(* Logix 5000 project; controller SolisPLC_Vlad_CGL1 vendor 1 type 14 code 226 rev 36.11; software revision 36.00 *)

TASK MainTask (continuous, watchdog 500 ms) : MainProgram, DataLink, Palletizer, Tutorials, Communication, SimulatedMachine_v1_0
TASK SafetyTask (periodic, rate 20 ms, priority 10, watchdog 20 ms, safety) : SafetyProgram

MODULES
   Local : vendor 1 type 14 code 226 (5069 0, rev 36.11)
      VFD_07 : PowerFlex 525-EENET (Ethernet 192.168.1.7, rev 1.3, Output RPI 20 ms)
END_MODULES

TYPE Asset_Data_v01_01 :
STRUCT
   machineState : INT;   // The state of the machine - 0 - Unknown State 1 - Running 2 - Stopped 3 - Stopped - Faulted 4 - Running - Starved 5 - Running - Backed-Up
   heartBeat : BOOL;   // A pulse which indicates that the communication with the machine is UP. The pulse is 1 sec ON / 1 sec OFF.
   currentProductionSpeed : INT;   // A count of finished products for the last hour.
END_STRUCT
END_TYPE

TYPE Motor_PF525_Params :
STRUCT
   Param_1_64 : INT[128];
   Param_65_128 : INT[128];
   Param_129_192 : INT[128];
   Param_193_256 : INT[128];
   Param_257_320 : INT[128];
   Param_321_384 : INT[128];
   Param_385_448 : INT[128];
   Param_449_512 : INT[128];
   Param_513_576 : INT[128];
   Param_577_640 : INT[128];
   Param_641_704 : INT[128];
   Param_705_768 : INT[128];
END_STRUCT
END_TYPE

TYPE UDT_MQTT_DINT :
STRUCT
   Message : DINT;
   Delay : DINT;
   Timer : TIMER;
   RawData : DINT;
   Delta : DINT;
   OldRawData : DINT;
END_STRUCT
END_TYPE

TYPE UDT_paramReadReqs :
STRUCT
   Param_1_64 : INT[128];
   Param_65_128 : INT[128];
   Param_129_192 : INT[128];
   Param_193_256 : INT[128];
   Param_257_320 : INT[128];
   Param_321_384 : INT[128];
   Param_385_448 : INT[128];
   Param_449_512 : INT[128];
   Param_513_576 : INT[128];
   Param_577_640 : INT[128];
   Param_641_704 : INT[128];
   Param_705_768 : INT[128];
END_STRUCT
END_TYPE

TYPE udtVariableSpeedMotor :
STRUCT
   Auto : BOOL;   // Auto Mode from RSView
   Interlock : BOOL;   // Pump Run Interlock
   Fault : BOOL;   // Pump Fault
   Start : BOOL;   // Manual Start from RSView
   Stop : BOOL;   // Manual Stop from RSView
   Run : BOOL;   // Drive Run Output Command
   Running : BOOL;   // Running Feedback
   LDS : BOOL;   // Local Disconnect Switch
   FwdCmd : BOOL;   // Run Drive Forward Request
   RevCmd : BOOL;   // Run Drive Reverse Request
   ClearFaults : BOOL;   // Drive Fault Reset Request
   Ready : BOOL;   // Drive Ready Feedback
   FwdAct : BOOL;   // Drive in Run Forward Mode
   RevAct : BOOL;   // Drive in Run Reverse Mode
   Alarm : BOOL;   // Drive Alarm
   DriveFault : BOOL;   // Drive Fault
   AtSpeed : BOOL;   // Drive is At Speed
   APerm : BOOL[32];   // Auto Run Permissive
   FaultTimer : TIMER;   // Start/Stop Timeout
   SpeedSP : REAL;   // Speed Setpoint from RSView
   SpeedSPmin : REAL;   // Speed Setpoint Minimum Limit
   SpeedSPmax : REAL;   // Speed Setpoint Maximum Limit
   SpeedAct : REAL;   // Actual Speed to RSView
   Status : DINT[5];
   Avl : BOOL[32];
   Name : Varchar40;
END_STRUCT
END_TYPE

TYPE Varchar40 :   // String Of 40 Characters
STRUCT
   LEN : DINT;
   DATA : SINT[40];
END_STRUCT
END_TYPE

ADD_ON_INSTRUCTION _AOI_Fah_to_Cel   (* revision 1.0 *)
VAR_INPUT
   Temperature_Fah : REAL; {required}
END_VAR
VAR_OUTPUT
   Temperature_Cel : REAL; {required}
END_VAR
VAR
   Placeholder : REAL; {access None}
   Placeholder1 : REAL; {access None}
END_VAR

ROUTINE Logic   (* ladder *)
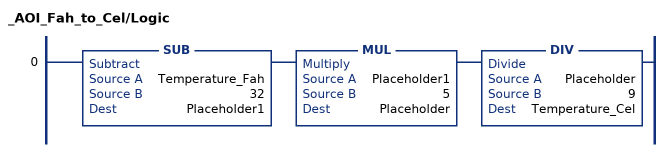
   0: SUB(Temperature_Fah,32,Placeholder1)MUL(Placeholder1,5,Placeholder)DIV(Placeholder,9,Temperature_Cel);
END_ROUTINE
END_ADD_ON_INSTRUCTION

ADD_ON_INSTRUCTION AOI_PF525_GetParam   (* revision 1.0 *)

ROUTINE Logic   (* ladder *)
END_ROUTINE
END_ADD_ON_INSTRUCTION

VAR_GLOBAL   (* controller tags *)
   BOOL_IN_0 : BOOL;
   BOOL_IN_1 : BOOL;   // System Stop PB
   BOOL_OUT_0 : BOOL;   // STATUS - System Running
   BOOL_OUT_1 : BOOL := 1;   // STATUS - System Stopped
   getParam : INT[10];
   M07_Params : Motor_PF525_Params := (Param_1_64[0] := 1, Param_1_64[2] := 2, Param_1_64[4] := 3, Param_1_64[6] := 4, Param_1_64[8] := 5, Param_1_64[9] := 329, Param_1_64[10] := 6, Param_1_64[11] := 2, Param_1_64[12] := 7, Param_1_64[13] := 73, Param_1_64[14] := 8, Param_1_64[15] := 4, Param_1_64[16] := 9, Param_1_64[17] := 73, Param_1_64[18] := 10, Param_1_64[20] := 11, Param_1_64[22] := 12, Param_1_64[23] := 155, Param_1_64[24] := 13, Param_1_64[25] := 1, Param_1_64[26] := 14, Param_1_64[28] := 15, Param_1_64[30] := 16, Param_1_64[32] := 17, Param_1_64[34] := 18, Param_1_64[36] := 19, Param_1_64[38] := 20, Param_1_64[40] := 21, Param_1_64[42] := 22, Param_1_64[44] := 23, Param_1_64[45] := 8, Param_1_64[46] := 24, Param_1_64[48] := 25, Param_1_64[50] := 26, Param_1_64[52] := 27, Param_1_64[53] := 30, Param_1_64[54] := 28, Param_1_64[55] := 53, Param_1_64[56] := 29, Param_1_64[57] := 7001, Param_1_64[58] := 30, Param_1_64[59] := 1, Param_1_64[60] := 31, Param_1_64[61] := 230, Param_1_64[62] := 32, Param_1_64[63] := 60, Param_1_64[64] := 33, Param_1_64[65] := 25, Param_1_64[66] := 34, Param_1_64[67] := 17, Param_1_64[68] := 35, Param_1_64[69] := 4, Param_1_64[70] := 36, Param_1_64[71] := 1750, Param_1_64[72] := 37, Param_1_64[73] := 40, Param_1_64[74] := 38, Param_1_64[76] := 39, Param_1_64[77] := 1, Param_1_64[78] := 40,
        Param_1_64[80] := 41, Param_1_64[81] := 1000, Param_1_64[82] := 42, Param_1_64[83] := 1000, Param_1_64[84] := 43, Param_1_64[86] := 44, Param_1_64[87] := 6000, Param_1_64[88] := 45, Param_1_64[90] := 46, Param_1_64[91] := 5, Param_1_64[92] := 47, Param_1_64[93] := 15, Param_1_64[94] := 48, Param_1_64[95] := 2, Param_1_64[96] := 49, Param_1_64[97] := 5, Param_1_64[98] := 50, Param_1_64[99] := 5, Param_1_64[100] := 51, Param_1_64[101] := 15, Param_1_64[102] := 52, Param_1_64[104] := 53, Param_1_64[106] := 54, Param_1_64[108] := 55, Param_1_64[110] := 56, Param_1_64[112] := 57, Param_1_64[114] := 58, Param_1_64[116] := 59, Param_1_64[118] := 60, Param_1_64[120] := 61, Param_1_64[122] := 62, Param_1_64[123] := 48, Param_1_64[124] := 63, Param_1_64[125] := 50, Param_1_64[126] := 64, Param_65_128[0] := 65, Param_65_128[2] := 66, Param_65_128[3] := 7, Param_65_128[4] := 67, Param_65_128[5] := 5, Param_65_128[6] := 68, Param_65_128[7] := 9, Param_65_128[8] := 69, Param_65_128[9] := 2, Param_65_128[10] := 70, Param_65_128[12] := 71, Param_65_128[14] := 72, Param_65_128[15] := 1, Param_65_128[16] := 73, Param_65_128[18] := 74, Param_65_128[20] := 75, Param_65_128[22] := 76, Param_65_128[24] := 77, Param_65_128[26] := 78, Param_65_128[28] := 79, Param_65_128[30] := 80, Param_65_128[32] := 81, Param_65_128[33] := 13, Param_65_128[34] := 82, Param_65_128[36] := 83,
        Param_65_128[38] := 84, Param_65_128[40] := 85, Param_65_128[42] := 86, Param_65_128[43] := 200, Param_65_128[44] := 87, Param_65_128[45] := 200, Param_65_128[46] := 88, Param_65_128[48] := 89, Param_65_128[49] := 100, Param_65_128[50] := 90, Param_65_128[52] := 91, Param_65_128[54] := 92, Param_65_128[55] := 1000, Param_65_128[56] := 93, Param_65_128[58] := 94, Param_65_128[60] := 95, Param_65_128[62] := 96, Param_65_128[63] := 1000, Param_65_128[64] := 97, Param_65_128[66] := 98, Param_65_128[68] := 99, Param_65_128[70] := 100, Param_65_128[72] := 101, Param_65_128[73] := 100, Param_65_128[74] := 102, Param_65_128[76] := 103, Param_65_128[77] := 150, Param_65_128[78] := 104, Param_65_128[80] := 105, Param_65_128[82] := 106, Param_65_128[84] := 107, Param_65_128[86] := 108, Param_65_128[88] := 109, Param_65_128[90] := 110, Param_65_128[92] := 111, Param_65_128[94] := 112, Param_65_128[96] := 113, Param_65_128[98] := 114, Param_65_128[100] := 115, Param_65_128[102] := 116, Param_65_128[104] := 117, Param_65_128[106] := 118, Param_65_128[108] := 119, Param_65_128[110] := 120, Param_65_128[112] := 121, Param_65_128[114] := 122, Param_65_128[116] := 123, Param_65_128[117] := 3, Param_65_128[118] := 124, Param_65_128[119] := 100, Param_65_128[120] := 125, Param_65_128[122] := 126, Param_65_128[123] := 50, Param_65_128[124] := 127, Param_65_128[126] := 128, Param_65_128[127] := 1, Param_129_192[0] := 129, Param_129_192[1] := 192, Param_129_192[2] := 130, Param_129_192[3] := 168,
        Param_129_192[4] := 131, Param_129_192[5] := 1, Param_129_192[6] := 132, Param_129_192[7] := 7, Param_129_192[8] := 133, Param_129_192[9] := 255, Param_129_192[10] := 134, Param_129_192[11] := 255, Param_129_192[12] := 135, Param_129_192[13] := 255, Param_129_192[14] := 136, Param_129_192[16] := 137, Param_129_192[18] := 138, Param_129_192[20] := 139, Param_129_192[22] := 140, Param_129_192[24] := 141, Param_129_192[26] := 142, Param_129_192[28] := 143, Param_129_192[30] := 144, Param_129_192[32] := 145, Param_129_192[34] := 146, Param_129_192[36] := 147, Param_129_192[38] := 148, Param_129_192[40] := 149, Param_129_192[42] := 150, Param_129_192[44] := 151, Param_129_192[46] := 152, Param_129_192[48] := 153, Param_129_192[49] := 82, Param_129_192[50] := 154, Param_129_192[52] := 155, Param_129_192[54] := 156, Param_129_192[56] := 157, Param_129_192[57] := 14, Param_129_192[58] := 158, Param_129_192[60] := 159, Param_129_192[62] := 160, Param_129_192[64] := 161, Param_129_192[66] := 162, Param_129_192[68] := 163, Param_129_192[70] := 164, Param_129_192[72] := 165, Param_129_192[74] := 166, Param_129_192[76] := 167, Param_129_192[78] := 168, Param_129_192[80] := 169, Param_129_192[82] := 170, Param_129_192[84] := 171, Param_129_192[85] := 2, Param_129_192[86] := 172, Param_129_192[87] := 3, Param_129_192[88] := 173, Param_129_192[89] := 4, Param_129_192[90] := 174, Param_129_192[91] := 5, Param_129_192[92] := 175, Param_129_192[94] := 176, Param_129_192[96] := 177, Param_129_192[98] := 178, Param_129_192[100] := 179,
        Param_129_192[102] := 180, Param_129_192[103] := 241, Param_129_192[104] := 181, Param_129_192[105] := 241, Param_129_192[106] := 182, Param_129_192[107] := 241, Param_129_192[108] := 183, Param_129_192[109] := 241, Param_129_192[110] := 184, Param_129_192[111] := 241, Param_129_192[112] := 185, Param_129_192[113] := 241, Param_129_192[114] := 186, Param_129_192[115] := 241, Param_129_192[116] := 187, Param_129_192[117] := 241, Param_129_192[118] := 188, Param_129_192[120] := 189, Param_129_192[122] := 190, Param_129_192[123] := 300, Param_129_192[124] := 191, Param_129_192[125] := 300, Param_129_192[126] := 192, Param_129_192[127] := 300, Param_193_256[0] := 193, Param_193_256[1] := 300, Param_193_256[2] := 194, Param_193_256[3] := 300, Param_193_256[4] := 195, Param_193_256[5] := 300, Param_193_256[6] := 196, Param_193_256[7] := 300, Param_193_256[8] := 197, Param_193_256[9] := 300, Param_193_256[10] := 198, Param_193_256[12] := 199, Param_193_256[14] := 200, Param_193_256[16] := 201, Param_193_256[18] := 202, Param_193_256[20] := 203, Param_193_256[22] := 204, Param_193_256[24] := 205, Param_193_256[26] := 206, Param_193_256[28] := 207, Param_193_256[30] := 208, Param_193_256[32] := 209, Param_193_256[34] := 210, Param_193_256[36] := 211, Param_193_256[38] := 212, Param_193_256[40] := 213, Param_193_256[42] := 214, Param_193_256[44] := 215, Param_193_256[46] := 216, Param_193_256[48] := 217, Param_193_256[50] := 218, Param_193_256[52] := 219, Param_193_256[54] := 220, Param_193_256[56] := 221, Param_193_256[58] := 222, Param_193_256[60] := 223,
        Param_193_256[62] := 224, Param_193_256[64] := 225, Param_193_256[66] := 226, Param_193_256[68] := 227, Param_193_256[70] := 228, Param_193_256[72] := 229, Param_193_256[74] := 230, Param_193_256[76] := 231, Param_193_256[78] := 232, Param_193_256[80] := 233, Param_193_256[82] := 234, Param_193_256[84] := 235, Param_193_256[86] := 236, Param_193_256[88] := 237, Param_193_256[90] := 238, Param_193_256[92] := 239, Param_193_256[94] := 240, Param_193_256[96] := 241, Param_193_256[98] := 242, Param_193_256[100] := 243, Param_193_256[102] := 244, Param_193_256[104] := 245, Param_193_256[106] := 246, Param_193_256[108] := 247, Param_193_256[110] := 248, Param_193_256[112] := 249, Param_193_256[114] := 250, Param_193_256[116] := 251, Param_193_256[118] := 252, Param_193_256[120] := 253, Param_193_256[122] := 254, Param_193_256[124] := 255, Param_193_256[126] := 256, Param_257_320[0] := 257, Param_257_320[2] := 258, Param_257_320[4] := 259, Param_257_320[6] := 260, Param_257_320[8] := 261, Param_257_320[10] := 262, Param_257_320[12] := 263, Param_257_320[14] := 264, Param_257_320[16] := 265, Param_257_320[18] := 266, Param_257_320[20] := 267, Param_257_320[22] := 268, Param_257_320[24] := 269, Param_257_320[26] := 270, Param_257_320[28] := 271, Param_257_320[30] := 272, Param_257_320[32] := 273, Param_257_320[34] := 274, Param_257_320[36] := 275, Param_257_320[38] := 276, Param_257_320[40] := 277, Param_257_320[42] := 278, Param_257_320[44] := 279, Param_257_320[46] := 280, Param_257_320[48] := 281, Param_257_320[50] := 282, Param_257_320[52] := 283,
        Param_257_320[54] := 284, Param_257_320[56] := 285, Param_257_320[58] := 286, Param_257_320[60] := 287, Param_257_320[62] := 288, Param_257_320[64] := 289, Param_257_320[66] := 290, Param_257_320[68] := 291, Param_257_320[70] := 292, Param_257_320[72] := 293, Param_257_320[74] := 294, Param_257_320[76] := 295, Param_257_320[78] := 296, Param_257_320[80] := 297, Param_257_320[82] := 298, Param_257_320[84] := 299, Param_257_320[86] := 300, Param_257_320[88] := 301, Param_257_320[90] := 302, Param_257_320[92] := 303, Param_257_320[94] := 304, Param_257_320[96] := 305, Param_257_320[98] := 306, Param_257_320[100] := 307, Param_257_320[102] := 308, Param_257_320[104] := 309, Param_257_320[106] := 310, Param_257_320[108] := 311, Param_257_320[110] := 312, Param_257_320[112] := 313, Param_257_320[114] := 314, Param_257_320[116] := 315, Param_257_320[118] := 316, Param_257_320[120] := 317, Param_257_320[122] := 318, Param_257_320[124] := 319, Param_257_320[126] := 320, Param_321_384[0] := 321, Param_321_384[2] := 322, Param_321_384[4] := 323, Param_321_384[6] := 324, Param_321_384[8] := 325, Param_321_384[10] := 326, Param_321_384[12] := 327, Param_321_384[14] := 328, Param_321_384[16] := 329, Param_321_384[18] := 330, Param_321_384[20] := 331, Param_321_384[22] := 332, Param_321_384[24] := 333, Param_321_384[26] := 334, Param_321_384[28] := 335, Param_321_384[30] := 336, Param_321_384[32] := 337, Param_321_384[34] := 338, Param_321_384[36] := 339, Param_321_384[38] := 340, Param_321_384[40] := 341, Param_321_384[42] := 342, Param_321_384[44] := 343,
        Param_321_384[46] := 344, Param_321_384[48] := 345, Param_321_384[50] := 346, Param_321_384[52] := 347, Param_321_384[54] := 348, Param_321_384[56] := 349, Param_321_384[58] := 350, Param_321_384[60] := 351, Param_321_384[62] := 352, Param_321_384[64] := 353, Param_321_384[66] := 354, Param_321_384[68] := 355, Param_321_384[70] := 356, Param_321_384[72] := 357, Param_321_384[74] := 358, Param_321_384[76] := 359, Param_321_384[78] := 360, Param_321_384[80] := 361, Param_321_384[82] := 362, Param_321_384[83] := 978, Param_321_384[84] := 363, Param_321_384[85] := 72, Param_321_384[86] := 364, Param_321_384[88] := 365, Param_321_384[90] := 366, Param_321_384[92] := 367, Param_321_384[93] := 1502, Param_321_384[94] := 368, Param_321_384[96] := 369, Param_321_384[98] := 370, Param_321_384[100] := 371, Param_321_384[102] := 372, Param_321_384[104] := 373, Param_321_384[106] := 374, Param_321_384[108] := 375, Param_321_384[110] := 376, Param_321_384[112] := 377, Param_321_384[114] := 378, Param_321_384[116] := 379, Param_321_384[118] := 380, Param_321_384[120] := 381, Param_321_384[122] := 382, Param_321_384[124] := 383, Param_321_384[126] := 384, Param_385_448[0] := 385, Param_385_448[2] := 386, Param_385_448[4] := 387, Param_385_448[5] := 5, Param_385_448[6] := 388, Param_385_448[8] := 389, Param_385_448[10] := 390, Param_385_448[12] := 391, Param_385_448[14] := 392, Param_385_448[16] := 393, Param_385_448[17] := 11264, Param_385_448[18] := 394, Param_385_448[19] := 1, Param_385_448[20] := 395, Param_385_448[22] := 396, Param_385_448[24] := 397,
        Param_385_448[26] := 398, Param_385_448[28] := 399, Param_385_448[30] := 400, Param_385_448[32] := 401, Param_385_448[34] := 402, Param_385_448[36] := 403, Param_385_448[38] := 404, Param_385_448[40] := 405, Param_385_448[42] := 406, Param_385_448[44] := 407, Param_385_448[46] := 408, Param_385_448[48] := 409, Param_385_448[50] := 410, Param_385_448[52] := 411, Param_385_448[53] := 500, Param_385_448[54] := 412, Param_385_448[55] := 1000, Param_385_448[56] := 413, Param_385_448[57] := 2000, Param_385_448[58] := 414, Param_385_448[59] := 3000, Param_385_448[60] := 415, Param_385_448[61] := 4000, Param_385_448[62] := 416, Param_385_448[63] := 5000, Param_385_448[64] := 417, Param_385_448[65] := 6000, Param_385_448[66] := 418, Param_385_448[67] := 6000, Param_385_448[68] := 419, Param_385_448[69] := 6000, Param_385_448[70] := 420, Param_385_448[71] := 6000, Param_385_448[72] := 421, Param_385_448[73] := 6000, Param_385_448[74] := 422, Param_385_448[75] := 6000, Param_385_448[76] := 423, Param_385_448[77] := 6000, Param_385_448[78] := 424, Param_385_448[79] := 6000, Param_385_448[80] := 425, Param_385_448[81] := 6000, Param_385_448[82] := 426, Param_385_448[83] := 6000, Param_385_448[84] := 427, Param_385_448[85] := 6000, Param_385_448[86] := 428, Param_385_448[87] := 1, Param_385_448[88] := 429, Param_385_448[90] := 430, Param_385_448[91] := 100, Param_385_448[92] := 431, Param_385_448[93] := 1000, Param_385_448[94] := 432, Param_385_448[95] := 1000, Param_385_448[96] := 433, Param_385_448[97] := 500, Param_385_448[98] := 434, Param_385_448[100] := 435,
        Param_385_448[101] := 1, Param_385_448[102] := 436, Param_385_448[104] := 437, Param_385_448[106] := 438, Param_385_448[107] := 1000, Param_385_448[108] := 439, Param_385_448[110] := 440, Param_385_448[111] := 40, Param_385_448[112] := 441, Param_385_448[114] := 442, Param_385_448[115] := 1000, Param_385_448[116] := 443, Param_385_448[117] := 1000, Param_385_448[118] := 444, Param_385_448[119] := 1000, Param_385_448[120] := 445, Param_385_448[121] := 1000, Param_385_448[122] := 446, Param_385_448[123] := 1000, Param_385_448[124] := 447, Param_385_448[125] := 1000, Param_385_448[126] := 448, Param_449_512[0] := 449, Param_449_512[2] := 450, Param_449_512[4] := 451, Param_449_512[6] := 452, Param_449_512[8] := 453, Param_449_512[10] := 454, Param_449_512[12] := 455, Param_449_512[14] := 456, Param_449_512[15] := 600, Param_449_512[16] := 457, Param_449_512[18] := 458, Param_449_512[20] := 459, Param_449_512[22] := 460, Param_449_512[24] := 461, Param_449_512[25] := 1, Param_449_512[26] := 462, Param_449_512[27] := 20, Param_449_512[28] := 463, Param_449_512[30] := 464, Param_449_512[32] := 465, Param_449_512[34] := 466, Param_449_512[36] := 467, Param_449_512[38] := 468, Param_449_512[39] := 600, Param_449_512[40] := 469, Param_449_512[42] := 470, Param_449_512[44] := 471, Param_449_512[46] := 472, Param_449_512[48] := 473, Param_449_512[49] := 1, Param_449_512[50] := 474, Param_449_512[51] := 20, Param_449_512[52] := 475, Param_449_512[54] := 476, Param_449_512[56] := 477, Param_449_512[58] := 478, Param_449_512[60] := 479, Param_449_512[62] := 480,
        Param_449_512[64] := 481, Param_449_512[66] := 482, Param_449_512[68] := 483, Param_449_512[69] := 1024, Param_449_512[70] := 484, Param_449_512[71] := 38, Param_449_512[72] := 485, Param_449_512[73] := 28, Param_449_512[74] := 486, Param_449_512[76] := 487, Param_449_512[78] := 488, Param_449_512[80] := 489, Param_449_512[82] := 490, Param_449_512[84] := 491, Param_449_512[86] := 492, Param_449_512[88] := 493, Param_449_512[90] := 494, Param_449_512[92] := 495, Param_449_512[93] := 3, Param_449_512[94] := 496, Param_449_512[95] := 87, Param_449_512[96] := 497, Param_449_512[97] := 87, Param_449_512[98] := 498, Param_449_512[100] := 499, Param_449_512[102] := 500, Param_449_512[104] := 501, Param_449_512[105] := 1150, Param_449_512[106] := 502, Param_449_512[107] := 1791, Param_449_512[108] := 503, Param_449_512[109] := 5321, Param_449_512[110] := 504, Param_449_512[111] := 1640, Param_449_512[112] := 505, Param_449_512[114] := 506, Param_449_512[116] := 507, Param_449_512[118] := 508, Param_449_512[120] := 509, Param_449_512[122] := 510, Param_449_512[123] := 833, Param_449_512[124] := 511, Param_449_512[125] := 10, Param_449_512[126] := 512, Param_449_512[127] := 1500, Param_513_576[0] := 513, Param_513_576[1] := 10, Param_513_576[2] := 514, Param_513_576[3] := 2000, Param_513_576[4] := 515, Param_513_576[5] := 10, Param_513_576[6] := 516, Param_513_576[8] := 517, Param_513_576[9] := 30, Param_513_576[10] := 518, Param_513_576[11] := 7, Param_513_576[12] := 519, Param_513_576[13] := 100, Param_513_576[14] := 520, Param_513_576[15] := 2,
        Param_513_576[16] := 521, Param_513_576[17] := 1000, Param_513_576[18] := 522, Param_513_576[19] := 100, Param_513_576[20] := 523, Param_513_576[21] := 1000, Param_513_576[22] := 524, Param_513_576[23] := 100, Param_513_576[24] := 525, Param_513_576[25] := 1000, Param_513_576[26] := 526, Param_513_576[27] := 100, Param_513_576[28] := 527, Param_513_576[29] := 350, Param_513_576[30] := 528, Param_513_576[31] := 300, Param_513_576[32] := 529, Param_513_576[33] := 7, Param_513_576[34] := 530, Param_513_576[35] := 8, Param_513_576[36] := 531, Param_513_576[37] := 25, Param_513_576[38] := 532, Param_513_576[39] := 250, Param_513_576[40] := 533, Param_513_576[41] := 150, Param_513_576[42] := 534, Param_513_576[43] := 230, Param_513_576[44] := 535, Param_513_576[46] := 536, Param_513_576[47] := 1024, Param_513_576[48] := 537, Param_513_576[49] := 64, Param_513_576[50] := 538, Param_513_576[51] := 20, Param_513_576[52] := 539, Param_513_576[53] := 5, Param_513_576[54] := 540, Param_513_576[56] := 541, Param_513_576[58] := 542, Param_513_576[59] := 10, Param_513_576[60] := 543, Param_513_576[62] := 544, Param_513_576[64] := 545, Param_513_576[66] := 546, Param_513_576[67] := 65, Param_513_576[68] := 547, Param_513_576[69] := 1, Param_513_576[70] := 548, Param_513_576[72] := 549, Param_513_576[74] := 550, Param_513_576[75] := 1, Param_513_576[76] := 551, Param_513_576[78] := 552, Param_513_576[80] := 553, Param_513_576[82] := 554, Param_513_576[84] := 555, Param_513_576[86] := 556, Param_513_576[87] := 2, Param_513_576[88] := 557,
        Param_513_576[90] := 558, Param_513_576[92] := 559, Param_513_576[93] := 4096, Param_513_576[94] := 560, Param_513_576[96] := 561, Param_513_576[98] := 562, Param_513_576[99] := 100, Param_513_576[100] := 563, Param_513_576[102] := 564, Param_513_576[103] := 100, Param_513_576[104] := 565, Param_513_576[105] := 8, Param_513_576[106] := 566, Param_513_576[107] := 30, Param_513_576[108] := 567, Param_513_576[110] := 568, Param_513_576[112] := 569, Param_513_576[114] := 570, Param_513_576[116] := 571, Param_513_576[118] := 572, Param_513_576[119] := 100, Param_513_576[120] := 573, Param_513_576[121] := 3, Param_513_576[122] := 574, Param_513_576[124] := 575, Param_513_576[126] := 576, Param_513_576[127] := 250, Param_577_640[0] := 577, Param_577_640[2] := 578, Param_577_640[4] := 579, Param_577_640[6] := 580, Param_577_640[8] := 581, Param_577_640[10] := 582, Param_577_640[11] := 45, Param_577_640[12] := 583, Param_577_640[13] := 40, Param_577_640[14] := 584, Param_577_640[15] := 250, Param_577_640[16] := 585, Param_577_640[17] := 40, Param_577_640[18] := 586, Param_577_640[20] := 587, Param_577_640[21] := 120, Param_577_640[22] := 588, Param_577_640[23] := 500, Param_577_640[24] := 589, Param_577_640[26] := 590, Param_577_640[27] := 1000, Param_577_640[28] := 591, Param_577_640[29] := 35, Param_577_640[30] := 592, Param_577_640[31] := 30, Param_577_640[32] := 593, Param_577_640[33] := 100, Param_577_640[34] := 594, Param_577_640[35] := 100, Param_577_640[36] := 595, Param_577_640[37] := 10, Param_577_640[38] := 596, Param_577_640[39] := 10,
        Param_577_640[40] := 597, Param_577_640[42] := 598, Param_577_640[44] := 599, Param_577_640[46] := 600, Param_577_640[48] := 601, Param_577_640[50] := 602, Param_577_640[52] := 603, Param_577_640[54] := 604, Param_577_640[55] := 4, Param_577_640[56] := 605, Param_577_640[58] := 606, Param_577_640[60] := 607, Param_577_640[62] := 608, Param_577_640[64] := 609, Param_577_640[66] := 610, Param_577_640[68] := 611, Param_577_640[69] := 967, Param_577_640[70] := 612, Param_577_640[71] := 166, Param_577_640[72] := 613, Param_577_640[73] := 140, Param_577_640[74] := 614, Param_577_640[75] := 92, Param_577_640[76] := 615, Param_577_640[78] := 616, Param_577_640[80] := 617, Param_577_640[82] := 618, Param_577_640[84] := 619, Param_577_640[86] := 620, Param_577_640[88] := 621, Param_577_640[89] := 452, Param_577_640[90] := 622, Param_577_640[91] := 154, Param_577_640[92] := 623, Param_577_640[93] := 472, Param_577_640[94] := 624, Param_577_640[95] := 566, Param_577_640[96] := 625, Param_577_640[98] := 626, Param_577_640[100] := 627, Param_577_640[102] := 628, Param_577_640[104] := 629, Param_577_640[106] := 630, Param_577_640[108] := 631, Param_577_640[110] := 632, Param_577_640[112] := 633, Param_577_640[114] := 634, Param_577_640[116] := 635, Param_577_640[118] := 636, Param_577_640[120] := 637, Param_577_640[122] := 638, Param_577_640[124] := 639, Param_577_640[126] := 640, Param_641_704[0] := 641, Param_641_704[2] := 642, Param_641_704[4] := 643, Param_641_704[6] := 644, Param_641_704[8] := 645, Param_641_704[10] := 646, Param_641_704[12] := 647,
        Param_641_704[14] := 648, Param_641_704[16] := 649, Param_641_704[18] := 650, Param_641_704[20] := 651, Param_641_704[21] := 330, Param_641_704[22] := 652, Param_641_704[23] := 184, Param_641_704[24] := 653, Param_641_704[25] := 331, Param_641_704[26] := 654, Param_641_704[27] := 184, Param_641_704[28] := 655, Param_641_704[30] := 656, Param_641_704[32] := 657, Param_641_704[34] := 658, Param_641_704[36] := 659, Param_641_704[38] := 660, Param_641_704[40] := 661, Param_641_704[41] := 2, Param_641_704[42] := 662, Param_641_704[43] := 2, Param_641_704[44] := 663, Param_641_704[45] := 2, Param_641_704[46] := 664, Param_641_704[47] := 2, Param_641_704[48] := 665, Param_641_704[50] := 666, Param_641_704[52] := 667, Param_641_704[54] := 668, Param_641_704[56] := 669, Param_641_704[58] := 670, Param_641_704[60] := 671, Param_641_704[62] := 672, Param_641_704[64] := 673, Param_641_704[66] := 674, Param_641_704[68] := 675, Param_641_704[70] := 676, Param_641_704[72] := 677, Param_641_704[74] := 678, Param_641_704[76] := 679, Param_641_704[78] := 680, Param_641_704[80] := 681, Param_641_704[81] := 100, Param_641_704[82] := 682, Param_641_704[84] := 683, Param_641_704[85] := 111, Param_641_704[86] := 684, Param_641_704[87] := 1, Param_641_704[88] := 685, Param_641_704[89] := 3, Param_641_704[90] := 686, Param_641_704[91] := 1, Param_641_704[92] := 687, Param_641_704[94] := 688, Param_641_704[95] := 29, Param_641_704[96] := 689, Param_641_704[97] := 156, Param_641_704[98] := 690, Param_641_704[99] := 233, Param_641_704[100] := 691,
        Param_641_704[101] := 106, Param_641_704[102] := 692, Param_641_704[103] := 186, Param_641_704[104] := 693, Param_641_704[105] := 192, Param_641_704[106] := 694, Param_641_704[107] := 168, Param_641_704[108] := 695, Param_641_704[109] := 1, Param_641_704[110] := 696, Param_641_704[111] := 7, Param_641_704[112] := 697, Param_641_704[113] := 255, Param_641_704[114] := 698, Param_641_704[115] := 255, Param_641_704[116] := 699, Param_641_704[117] := 255, Param_641_704[118] := 700, Param_641_704[120] := 701, Param_641_704[122] := 702, Param_641_704[124] := 703, Param_641_704[126] := 704, Param_705_768[0] := 705, Param_705_768[1] := 1, Param_705_768[2] := 706, Param_705_768[4] := 707, Param_705_768[5] := 1549, Param_705_768[6] := 708, Param_705_768[8] := 709, Param_705_768[10] := 710, Param_705_768[12] := 711, Param_705_768[14] := 712, Param_705_768[16] := 713, Param_705_768[18] := 714, Param_705_768[20] := 715, Param_705_768[22] := 716, Param_705_768[24] := 717, Param_705_768[26] := 718, Param_705_768[28] := 719, Param_705_768[30] := 720, Param_705_768[32] := 721, Param_705_768[34] := 722, Param_705_768[36] := 723, Param_705_768[38] := 724, Param_705_768[40] := 725, Param_705_768[42] := 726, Param_705_768[43] := -22401, Param_705_768[44] := 727, Param_705_768[46] := 728, Param_705_768[47] := -12404, Param_705_768[48] := 729, Param_705_768[50] := 730, Param_705_768[52] := 731, Param_705_768[54] := -32036, Param_705_768[55] := 22, Param_705_768[56] := -32035, Param_705_768[57] := 22, Param_705_768[58] := -32034, Param_705_768[59] := 22, Param_705_768[60] := -32033,
        Param_705_768[61] := 22, Param_705_768[62] := -32032, Param_705_768[63] := 22, Param_705_768[64] := -32031, Param_705_768[65] := 22, Param_705_768[66] := -32030, Param_705_768[67] := 22, Param_705_768[68] := -32029, Param_705_768[69] := 22, Param_705_768[70] := -32028, Param_705_768[71] := 22, Param_705_768[72] := -32027, Param_705_768[73] := 22, Param_705_768[74] := -32026, Param_705_768[75] := 22, Param_705_768[76] := -32025, Param_705_768[77] := 22, Param_705_768[78] := -32024, Param_705_768[79] := 22, Param_705_768[80] := -32023, Param_705_768[81] := 22, Param_705_768[82] := -32022, Param_705_768[83] := 22, Param_705_768[84] := -32021, Param_705_768[85] := 22, Param_705_768[86] := -32020, Param_705_768[87] := 22, Param_705_768[88] := -32019, Param_705_768[89] := 22, Param_705_768[90] := -32018, Param_705_768[91] := 22, Param_705_768[92] := -32017, Param_705_768[93] := 22, Param_705_768[94] := -32016, Param_705_768[95] := 22, Param_705_768[96] := -32015, Param_705_768[97] := 22, Param_705_768[98] := -32014, Param_705_768[99] := 22, Param_705_768[100] := -32013, Param_705_768[101] := 22, Param_705_768[102] := -32012, Param_705_768[103] := 22, Param_705_768[104] := -32011, Param_705_768[105] := 22, Param_705_768[106] := -32010, Param_705_768[107] := 22, Param_705_768[108] := -32009, Param_705_768[109] := 22, Param_705_768[110] := -32008, Param_705_768[111] := 22, Param_705_768[112] := -32007, Param_705_768[113] := 22, Param_705_768[114] := -32006, Param_705_768[115] := 22, Param_705_768[116] := -32005, Param_705_768[117] := 22, Param_705_768[118] := -32004, Param_705_768[119] := 22, Param_705_768[120] := -32003,
        Param_705_768[121] := 22, Param_705_768[122] := -32002, Param_705_768[123] := 22, Param_705_768[124] := -32001, Param_705_768[125] := 22, Param_705_768[126] := -32000, Param_705_768[127] := 22);
   M07_readReq : INT[20] := ([0] := 129, [2] := 130, [4] := 131, [6] := 132, [8] := 132);
   M07_readRes : INT[20] := ([0] := 129, [1] := 192, [2] := 130, [3] := 168, [4] := 131, [5] := 1, [6] := 132, [7] := 7, [8] := 132, [9] := 7);
   motorReadReqs : UDT_paramReadReqs := (Param_1_64[0] := 1, Param_1_64[2] := 2, Param_1_64[4] := 3, Param_1_64[6] := 4, Param_1_64[8] := 5, Param_1_64[10] := 6, Param_1_64[12] := 7, Param_1_64[14] := 8, Param_1_64[16] := 9, Param_1_64[18] := 10, Param_1_64[20] := 11, Param_1_64[22] := 12, Param_1_64[24] := 13, Param_1_64[26] := 14, Param_1_64[28] := 15, Param_1_64[30] := 16, Param_1_64[32] := 17, Param_1_64[34] := 18, Param_1_64[36] := 19, Param_1_64[38] := 20, Param_1_64[40] := 21, Param_1_64[42] := 22, Param_1_64[44] := 23, Param_1_64[46] := 24, Param_1_64[48] := 25, Param_1_64[50] := 26, Param_1_64[52] := 27, Param_1_64[54] := 28, Param_1_64[56] := 29, Param_1_64[58] := 30, Param_1_64[60] := 31, Param_1_64[62] := 32, Param_1_64[64] := 33, Param_1_64[66] := 34, Param_1_64[68] := 35, Param_1_64[70] := 36, Param_1_64[72] := 37, Param_1_64[74] := 38, Param_1_64[76] := 39, Param_1_64[78] := 40, Param_1_64[80] := 41, Param_1_64[82] := 42, Param_1_64[84] := 43, Param_1_64[86] := 44, Param_1_64[88] := 45, Param_1_64[90] := 46, Param_1_64[92] := 47, Param_1_64[94] := 48, Param_1_64[96] := 49, Param_1_64[98] := 50, Param_1_64[100] := 51, Param_1_64[102] := 52, Param_1_64[104] := 53, Param_1_64[106] := 54, Param_1_64[108] := 55, Param_1_64[110] := 56, Param_1_64[112] := 57, Param_1_64[114] := 58, Param_1_64[116] := 59, Param_1_64[118] := 60,
        Param_1_64[120] := 61, Param_1_64[122] := 62, Param_1_64[124] := 63, Param_1_64[126] := 64, Param_65_128[0] := 65, Param_65_128[2] := 66, Param_65_128[4] := 67, Param_65_128[6] := 68, Param_65_128[8] := 69, Param_65_128[10] := 70, Param_65_128[12] := 71, Param_65_128[14] := 72, Param_65_128[16] := 73, Param_65_128[18] := 74, Param_65_128[20] := 75, Param_65_128[22] := 76, Param_65_128[24] := 77, Param_65_128[26] := 78, Param_65_128[28] := 79, Param_65_128[30] := 80, Param_65_128[32] := 81, Param_65_128[34] := 82, Param_65_128[36] := 83, Param_65_128[38] := 84, Param_65_128[40] := 85, Param_65_128[42] := 86, Param_65_128[44] := 87, Param_65_128[46] := 88, Param_65_128[48] := 89, Param_65_128[50] := 90, Param_65_128[52] := 91, Param_65_128[54] := 92, Param_65_128[56] := 93, Param_65_128[58] := 94, Param_65_128[60] := 95, Param_65_128[62] := 96, Param_65_128[64] := 97, Param_65_128[66] := 98, Param_65_128[68] := 99, Param_65_128[70] := 100, Param_65_128[72] := 101, Param_65_128[74] := 102, Param_65_128[76] := 103, Param_65_128[78] := 104, Param_65_128[80] := 105, Param_65_128[82] := 106, Param_65_128[84] := 107, Param_65_128[86] := 108, Param_65_128[88] := 109, Param_65_128[90] := 110, Param_65_128[92] := 111, Param_65_128[94] := 112, Param_65_128[96] := 113, Param_65_128[98] := 114, Param_65_128[100] := 115, Param_65_128[102] := 116, Param_65_128[104] := 117, Param_65_128[106] := 118, Param_65_128[108] := 119, Param_65_128[110] := 120,
        Param_65_128[112] := 121, Param_65_128[114] := 122, Param_65_128[116] := 123, Param_65_128[118] := 124, Param_65_128[120] := 125, Param_65_128[122] := 126, Param_65_128[124] := 127, Param_65_128[126] := 128, Param_129_192[0] := 129, Param_129_192[2] := 130, Param_129_192[4] := 131, Param_129_192[6] := 132, Param_129_192[8] := 133, Param_129_192[10] := 134, Param_129_192[12] := 135, Param_129_192[14] := 136, Param_129_192[16] := 137, Param_129_192[18] := 138, Param_129_192[20] := 139, Param_129_192[22] := 140, Param_129_192[24] := 141, Param_129_192[26] := 142, Param_129_192[28] := 143, Param_129_192[30] := 144, Param_129_192[32] := 145, Param_129_192[34] := 146, Param_129_192[36] := 147, Param_129_192[38] := 148, Param_129_192[40] := 149, Param_129_192[42] := 150, Param_129_192[44] := 151, Param_129_192[46] := 152, Param_129_192[48] := 153, Param_129_192[50] := 154, Param_129_192[52] := 155, Param_129_192[54] := 156, Param_129_192[56] := 157, Param_129_192[58] := 158, Param_129_192[60] := 159, Param_129_192[62] := 160, Param_129_192[64] := 161, Param_129_192[66] := 162, Param_129_192[68] := 163, Param_129_192[70] := 164, Param_129_192[72] := 165, Param_129_192[74] := 166, Param_129_192[76] := 167, Param_129_192[78] := 168, Param_129_192[80] := 169, Param_129_192[82] := 170, Param_129_192[84] := 171, Param_129_192[86] := 172, Param_129_192[88] := 173, Param_129_192[90] := 174, Param_129_192[92] := 175, Param_129_192[94] := 176, Param_129_192[96] := 177, Param_129_192[98] := 178, Param_129_192[100] := 179, Param_129_192[102] := 180,
        Param_129_192[104] := 181, Param_129_192[106] := 182, Param_129_192[108] := 183, Param_129_192[110] := 184, Param_129_192[112] := 185, Param_129_192[114] := 186, Param_129_192[116] := 187, Param_129_192[118] := 188, Param_129_192[120] := 189, Param_129_192[122] := 190, Param_129_192[124] := 191, Param_129_192[126] := 192, Param_193_256[0] := 193, Param_193_256[2] := 194, Param_193_256[4] := 195, Param_193_256[6] := 196, Param_193_256[8] := 197, Param_193_256[10] := 198, Param_193_256[12] := 199, Param_193_256[14] := 200, Param_193_256[16] := 201, Param_193_256[18] := 202, Param_193_256[20] := 203, Param_193_256[22] := 204, Param_193_256[24] := 205, Param_193_256[26] := 206, Param_193_256[28] := 207, Param_193_256[30] := 208, Param_193_256[32] := 209, Param_193_256[34] := 210, Param_193_256[36] := 211, Param_193_256[38] := 212, Param_193_256[40] := 213, Param_193_256[42] := 214, Param_193_256[44] := 215, Param_193_256[46] := 216, Param_193_256[48] := 217, Param_193_256[50] := 218, Param_193_256[52] := 219, Param_193_256[54] := 220, Param_193_256[56] := 221, Param_193_256[58] := 222, Param_193_256[60] := 223, Param_193_256[62] := 224, Param_193_256[64] := 225, Param_193_256[66] := 226, Param_193_256[68] := 227, Param_193_256[70] := 228, Param_193_256[72] := 229, Param_193_256[74] := 230, Param_193_256[76] := 231, Param_193_256[78] := 232, Param_193_256[80] := 233, Param_193_256[82] := 234, Param_193_256[84] := 235, Param_193_256[86] := 236, Param_193_256[88] := 237, Param_193_256[90] := 238, Param_193_256[92] := 239, Param_193_256[94] := 240,
        Param_193_256[96] := 241, Param_193_256[98] := 242, Param_193_256[100] := 243, Param_193_256[102] := 244, Param_193_256[104] := 245, Param_193_256[106] := 246, Param_193_256[108] := 247, Param_193_256[110] := 248, Param_193_256[112] := 249, Param_193_256[114] := 250, Param_193_256[116] := 251, Param_193_256[118] := 252, Param_193_256[120] := 253, Param_193_256[122] := 254, Param_193_256[124] := 255, Param_193_256[126] := 256, Param_257_320[0] := 257, Param_257_320[2] := 258, Param_257_320[4] := 259, Param_257_320[6] := 260, Param_257_320[8] := 261, Param_257_320[10] := 262, Param_257_320[12] := 263, Param_257_320[14] := 264, Param_257_320[16] := 265, Param_257_320[18] := 266, Param_257_320[20] := 267, Param_257_320[22] := 268, Param_257_320[24] := 269, Param_257_320[26] := 270, Param_257_320[28] := 271, Param_257_320[30] := 272, Param_257_320[32] := 273, Param_257_320[34] := 274, Param_257_320[36] := 275, Param_257_320[38] := 276, Param_257_320[40] := 277, Param_257_320[42] := 278, Param_257_320[44] := 279, Param_257_320[46] := 280, Param_257_320[48] := 281, Param_257_320[50] := 282, Param_257_320[52] := 283, Param_257_320[54] := 284, Param_257_320[56] := 285, Param_257_320[58] := 286, Param_257_320[60] := 287, Param_257_320[62] := 288, Param_257_320[64] := 289, Param_257_320[66] := 290, Param_257_320[68] := 291, Param_257_320[70] := 292, Param_257_320[72] := 293, Param_257_320[74] := 294, Param_257_320[76] := 295, Param_257_320[78] := 296, Param_257_320[80] := 297, Param_257_320[82] := 298, Param_257_320[84] := 299, Param_257_320[86] := 300,
        Param_257_320[88] := 301, Param_257_320[90] := 302, Param_257_320[92] := 303, Param_257_320[94] := 304, Param_257_320[96] := 305, Param_257_320[98] := 306, Param_257_320[100] := 307, Param_257_320[102] := 308, Param_257_320[104] := 309, Param_257_320[106] := 310, Param_257_320[108] := 311, Param_257_320[110] := 312, Param_257_320[112] := 313, Param_257_320[114] := 314, Param_257_320[116] := 315, Param_257_320[118] := 316, Param_257_320[120] := 317, Param_257_320[122] := 318, Param_257_320[124] := 319, Param_257_320[126] := 320, Param_321_384[0] := 321, Param_321_384[2] := 322, Param_321_384[4] := 323, Param_321_384[6] := 324, Param_321_384[8] := 325, Param_321_384[10] := 326, Param_321_384[12] := 327, Param_321_384[14] := 328, Param_321_384[16] := 329, Param_321_384[18] := 330, Param_321_384[20] := 331, Param_321_384[22] := 332, Param_321_384[24] := 333, Param_321_384[26] := 334, Param_321_384[28] := 335, Param_321_384[30] := 336, Param_321_384[32] := 337, Param_321_384[34] := 338, Param_321_384[36] := 339, Param_321_384[38] := 340, Param_321_384[40] := 341, Param_321_384[42] := 342, Param_321_384[44] := 343, Param_321_384[46] := 344, Param_321_384[48] := 345, Param_321_384[50] := 346, Param_321_384[52] := 347, Param_321_384[54] := 348, Param_321_384[56] := 349, Param_321_384[58] := 350, Param_321_384[60] := 351, Param_321_384[62] := 352, Param_321_384[64] := 353, Param_321_384[66] := 354, Param_321_384[68] := 355, Param_321_384[70] := 356, Param_321_384[72] := 357, Param_321_384[74] := 358, Param_321_384[76] := 359, Param_321_384[78] := 360,
        Param_321_384[80] := 361, Param_321_384[82] := 362, Param_321_384[84] := 363, Param_321_384[86] := 364, Param_321_384[88] := 365, Param_321_384[90] := 366, Param_321_384[92] := 367, Param_321_384[94] := 368, Param_321_384[96] := 369, Param_321_384[98] := 370, Param_321_384[100] := 371, Param_321_384[102] := 372, Param_321_384[104] := 373, Param_321_384[106] := 374, Param_321_384[108] := 375, Param_321_384[110] := 376, Param_321_384[112] := 377, Param_321_384[114] := 378, Param_321_384[116] := 379, Param_321_384[118] := 380, Param_321_384[120] := 381, Param_321_384[122] := 382, Param_321_384[124] := 383, Param_321_384[126] := 384, Param_385_448[0] := 385, Param_385_448[2] := 386, Param_385_448[4] := 387, Param_385_448[6] := 388, Param_385_448[8] := 389, Param_385_448[10] := 390, Param_385_448[12] := 391, Param_385_448[14] := 392, Param_385_448[16] := 393, Param_385_448[18] := 394, Param_385_448[20] := 395, Param_385_448[22] := 396, Param_385_448[24] := 397, Param_385_448[26] := 398, Param_385_448[28] := 399, Param_385_448[30] := 400, Param_385_448[32] := 401, Param_385_448[34] := 402, Param_385_448[36] := 403, Param_385_448[38] := 404, Param_385_448[40] := 405, Param_385_448[42] := 406, Param_385_448[44] := 407, Param_385_448[46] := 408, Param_385_448[48] := 409, Param_385_448[50] := 410, Param_385_448[52] := 411, Param_385_448[54] := 412, Param_385_448[56] := 413, Param_385_448[58] := 414, Param_385_448[60] := 415, Param_385_448[62] := 416, Param_385_448[64] := 417, Param_385_448[66] := 418, Param_385_448[68] := 419, Param_385_448[70] := 420,
        Param_385_448[72] := 421, Param_385_448[74] := 422, Param_385_448[76] := 423, Param_385_448[78] := 424, Param_385_448[80] := 425, Param_385_448[82] := 426, Param_385_448[84] := 427, Param_385_448[86] := 428, Param_385_448[88] := 429, Param_385_448[90] := 430, Param_385_448[92] := 431, Param_385_448[94] := 432, Param_385_448[96] := 433, Param_385_448[98] := 434, Param_385_448[100] := 435, Param_385_448[102] := 436, Param_385_448[104] := 437, Param_385_448[106] := 438, Param_385_448[108] := 439, Param_385_448[110] := 440, Param_385_448[112] := 441, Param_385_448[114] := 442, Param_385_448[116] := 443, Param_385_448[118] := 444, Param_385_448[120] := 445, Param_385_448[122] := 446, Param_385_448[124] := 447, Param_385_448[126] := 448, Param_449_512[0] := 449, Param_449_512[2] := 450, Param_449_512[4] := 451, Param_449_512[6] := 452, Param_449_512[8] := 453, Param_449_512[10] := 454, Param_449_512[12] := 455, Param_449_512[14] := 456, Param_449_512[16] := 457, Param_449_512[18] := 458, Param_449_512[20] := 459, Param_449_512[22] := 460, Param_449_512[24] := 461, Param_449_512[26] := 462, Param_449_512[28] := 463, Param_449_512[30] := 464, Param_449_512[32] := 465, Param_449_512[34] := 466, Param_449_512[36] := 467, Param_449_512[38] := 468, Param_449_512[40] := 469, Param_449_512[42] := 470, Param_449_512[44] := 471, Param_449_512[46] := 472, Param_449_512[48] := 473, Param_449_512[50] := 474, Param_449_512[52] := 475, Param_449_512[54] := 476, Param_449_512[56] := 477, Param_449_512[58] := 478, Param_449_512[60] := 479, Param_449_512[62] := 480,
        Param_449_512[64] := 481, Param_449_512[66] := 482, Param_449_512[68] := 483, Param_449_512[70] := 484, Param_449_512[72] := 485, Param_449_512[74] := 486, Param_449_512[76] := 487, Param_449_512[78] := 488, Param_449_512[80] := 489, Param_449_512[82] := 490, Param_449_512[84] := 491, Param_449_512[86] := 492, Param_449_512[88] := 493, Param_449_512[90] := 494, Param_449_512[92] := 495, Param_449_512[94] := 496, Param_449_512[96] := 497, Param_449_512[98] := 498, Param_449_512[100] := 499, Param_449_512[102] := 500, Param_449_512[104] := 501, Param_449_512[106] := 502, Param_449_512[108] := 503, Param_449_512[110] := 504, Param_449_512[112] := 505, Param_449_512[114] := 506, Param_449_512[116] := 507, Param_449_512[118] := 508, Param_449_512[120] := 509, Param_449_512[122] := 510, Param_449_512[124] := 511, Param_449_512[126] := 512, Param_513_576[0] := 513, Param_513_576[2] := 514, Param_513_576[4] := 515, Param_513_576[6] := 516, Param_513_576[8] := 517, Param_513_576[10] := 518, Param_513_576[12] := 519, Param_513_576[14] := 520, Param_513_576[16] := 521, Param_513_576[18] := 522, Param_513_576[20] := 523, Param_513_576[22] := 524, Param_513_576[24] := 525, Param_513_576[26] := 526, Param_513_576[28] := 527, Param_513_576[30] := 528, Param_513_576[32] := 529, Param_513_576[34] := 530, Param_513_576[36] := 531, Param_513_576[38] := 532, Param_513_576[40] := 533, Param_513_576[42] := 534, Param_513_576[44] := 535, Param_513_576[46] := 536, Param_513_576[48] := 537, Param_513_576[50] := 538, Param_513_576[52] := 539, Param_513_576[54] := 540,
        Param_513_576[56] := 541, Param_513_576[58] := 542, Param_513_576[60] := 543, Param_513_576[62] := 544, Param_513_576[64] := 545, Param_513_576[66] := 546, Param_513_576[68] := 547, Param_513_576[70] := 548, Param_513_576[72] := 549, Param_513_576[74] := 550, Param_513_576[76] := 551, Param_513_576[78] := 552, Param_513_576[80] := 553, Param_513_576[82] := 554, Param_513_576[84] := 555, Param_513_576[86] := 556, Param_513_576[88] := 557, Param_513_576[90] := 558, Param_513_576[92] := 559, Param_513_576[94] := 560, Param_513_576[96] := 561, Param_513_576[98] := 562, Param_513_576[100] := 563, Param_513_576[102] := 564, Param_513_576[104] := 565, Param_513_576[106] := 566, Param_513_576[108] := 567, Param_513_576[110] := 568, Param_513_576[112] := 569, Param_513_576[114] := 570, Param_513_576[116] := 571, Param_513_576[118] := 572, Param_513_576[120] := 573, Param_513_576[122] := 574, Param_513_576[124] := 575, Param_513_576[126] := 576, Param_577_640[0] := 577, Param_577_640[2] := 578, Param_577_640[4] := 579, Param_577_640[6] := 580, Param_577_640[8] := 581, Param_577_640[10] := 582, Param_577_640[12] := 583, Param_577_640[14] := 584, Param_577_640[16] := 585, Param_577_640[18] := 586, Param_577_640[20] := 587, Param_577_640[22] := 588, Param_577_640[24] := 589, Param_577_640[26] := 590, Param_577_640[28] := 591, Param_577_640[30] := 592, Param_577_640[32] := 593, Param_577_640[34] := 594, Param_577_640[36] := 595, Param_577_640[38] := 596, Param_577_640[40] := 597, Param_577_640[42] := 598, Param_577_640[44] := 599, Param_577_640[46] := 600,
        Param_577_640[48] := 601, Param_577_640[50] := 602, Param_577_640[52] := 603, Param_577_640[54] := 604, Param_577_640[56] := 605, Param_577_640[58] := 606, Param_577_640[60] := 607, Param_577_640[62] := 608, Param_577_640[64] := 609, Param_577_640[66] := 610, Param_577_640[68] := 611, Param_577_640[70] := 612, Param_577_640[72] := 613, Param_577_640[74] := 614, Param_577_640[76] := 615, Param_577_640[78] := 616, Param_577_640[80] := 617, Param_577_640[82] := 618, Param_577_640[84] := 619, Param_577_640[86] := 620, Param_577_640[88] := 621, Param_577_640[90] := 622, Param_577_640[92] := 623, Param_577_640[94] := 624, Param_577_640[96] := 625, Param_577_640[98] := 626, Param_577_640[100] := 627, Param_577_640[102] := 628, Param_577_640[104] := 629, Param_577_640[106] := 630, Param_577_640[108] := 631, Param_577_640[110] := 632, Param_577_640[112] := 633, Param_577_640[114] := 634, Param_577_640[116] := 635, Param_577_640[118] := 636, Param_577_640[120] := 637, Param_577_640[122] := 638, Param_577_640[124] := 639, Param_577_640[126] := 640, Param_641_704[0] := 641, Param_641_704[2] := 642, Param_641_704[4] := 643, Param_641_704[6] := 644, Param_641_704[8] := 645, Param_641_704[10] := 646, Param_641_704[12] := 647, Param_641_704[14] := 648, Param_641_704[16] := 649, Param_641_704[18] := 650, Param_641_704[20] := 651, Param_641_704[22] := 652, Param_641_704[24] := 653, Param_641_704[26] := 654, Param_641_704[28] := 655, Param_641_704[30] := 656, Param_641_704[32] := 657, Param_641_704[34] := 658, Param_641_704[36] := 659, Param_641_704[38] := 660,
        Param_641_704[40] := 661, Param_641_704[42] := 662, Param_641_704[44] := 663, Param_641_704[46] := 664, Param_641_704[48] := 665, Param_641_704[50] := 666, Param_641_704[52] := 667, Param_641_704[54] := 668, Param_641_704[56] := 669, Param_641_704[58] := 670, Param_641_704[60] := 671, Param_641_704[62] := 672, Param_641_704[64] := 673, Param_641_704[66] := 674, Param_641_704[68] := 675, Param_641_704[70] := 676, Param_641_704[72] := 677, Param_641_704[74] := 678, Param_641_704[76] := 679, Param_641_704[78] := 680, Param_641_704[80] := 681, Param_641_704[82] := 682, Param_641_704[84] := 683, Param_641_704[86] := 684, Param_641_704[88] := 685, Param_641_704[90] := 686, Param_641_704[92] := 687, Param_641_704[94] := 688, Param_641_704[96] := 689, Param_641_704[98] := 690, Param_641_704[100] := 691, Param_641_704[102] := 692, Param_641_704[104] := 693, Param_641_704[106] := 694, Param_641_704[108] := 695, Param_641_704[110] := 696, Param_641_704[112] := 697, Param_641_704[114] := 698, Param_641_704[116] := 699, Param_641_704[118] := 700, Param_641_704[120] := 701, Param_641_704[122] := 702, Param_641_704[124] := 703, Param_641_704[126] := 704, Param_705_768[0] := 705, Param_705_768[2] := 706, Param_705_768[4] := 707, Param_705_768[6] := 708, Param_705_768[8] := 709, Param_705_768[10] := 710, Param_705_768[12] := 711, Param_705_768[14] := 712, Param_705_768[16] := 713, Param_705_768[18] := 714, Param_705_768[20] := 715, Param_705_768[22] := 716, Param_705_768[24] := 717, Param_705_768[26] := 718, Param_705_768[28] := 719, Param_705_768[30] := 720,
        Param_705_768[32] := 721, Param_705_768[34] := 722, Param_705_768[36] := 723, Param_705_768[38] := 724, Param_705_768[40] := 725, Param_705_768[42] := 726, Param_705_768[44] := 727, Param_705_768[46] := 728, Param_705_768[48] := 729, Param_705_768[50] := 730, Param_705_768[52] := 731, Param_705_768[54] := 732, Param_705_768[56] := 733, Param_705_768[58] := 734, Param_705_768[60] := 735, Param_705_768[62] := 736, Param_705_768[64] := 737, Param_705_768[66] := 738, Param_705_768[68] := 739, Param_705_768[70] := 740, Param_705_768[72] := 741, Param_705_768[74] := 742, Param_705_768[76] := 743, Param_705_768[78] := 744, Param_705_768[80] := 745, Param_705_768[82] := 746, Param_705_768[84] := 747, Param_705_768[86] := 748, Param_705_768[88] := 749, Param_705_768[90] := 750, Param_705_768[92] := 751, Param_705_768[94] := 752, Param_705_768[96] := 753, Param_705_768[98] := 754, Param_705_768[100] := 755, Param_705_768[102] := 756, Param_705_768[104] := 757, Param_705_768[106] := 758, Param_705_768[108] := 759, Param_705_768[110] := 760, Param_705_768[112] := 761, Param_705_768[114] := 762, Param_705_768[116] := 763, Param_705_768[118] := 764, Param_705_768[120] := 765, Param_705_768[122] := 766, Param_705_768[124] := 767, Param_705_768[126] := 768);
   MQTT_OUT : UDT_MQTT_DINT[100] := ([0].Message := 2380, [0].Timer.EN := 1, [0].Timer.TT := 1, [0].RawData := 2380, [0].OldRawData := 2380, [1].Message := 9, [1].Timer.EN := 1, [1].Timer.TT := 1, [1].RawData := 9, [1].OldRawData := 9, [2].Message := 16, [2].Timer.EN := 1, [2].Timer.TT := 1, [2].RawData := 16, [2].OldRawData := 16, [3].Message := 1361, [3].Delay := 1000, [3].Timer.PRE := 1000, [3].Timer.ACC := 148, [3].Timer.EN := 1, [3].Timer.TT := 1, [3].RawData := 1509, [3].Delta := 1000, [3].OldRawData := 1361, [4].Delay := 1000, [4].Timer.PRE := 1000, [4].Timer.ACC := 509, [4].Timer.EN := 1, [4].Timer.TT := 1, [4].Delta := 1000, [5].Timer.EN := 1, [5].Timer.TT := 1, [6].Timer.EN := 1, [6].Timer.TT := 1, [7].Timer.EN := 1, [7].Timer.TT := 1, [8].Timer.EN := 1, [8].Timer.TT := 1, [9].Timer.EN := 1, [9].Timer.TT := 1, [10].Timer.EN := 1, [10].Timer.TT := 1, [11].Timer.EN := 1, [11].Timer.TT := 1, [12].Timer.EN := 1, [12].Timer.TT := 1, [13].Timer.EN := 1, [13].Timer.TT := 1, [14].Timer.EN := 1, [14].Timer.TT := 1, [15].Timer.EN := 1, [15].Timer.TT := 1, [16].Timer.EN := 1, [16].Timer.TT := 1, [17].Timer.EN := 1, [17].Timer.TT := 1, [18].Timer.EN := 1, [18].Timer.TT := 1, [19].Timer.EN := 1, [19].Timer.TT := 1,
        [20].Timer.EN := 1, [20].Timer.TT := 1, [21].Timer.EN := 1, [21].Timer.TT := 1, [22].Timer.EN := 1, [22].Timer.TT := 1, [23].Timer.EN := 1, [23].Timer.TT := 1, [24].Timer.EN := 1, [24].Timer.TT := 1, [25].Timer.EN := 1, [25].Timer.TT := 1, [26].Timer.EN := 1, [26].Timer.TT := 1, [27].Timer.EN := 1, [27].Timer.TT := 1, [28].Timer.EN := 1, [28].Timer.TT := 1, [29].Timer.EN := 1, [29].Timer.TT := 1, [30].Timer.EN := 1, [30].Timer.TT := 1, [31].Timer.EN := 1, [31].Timer.TT := 1, [32].Timer.EN := 1, [32].Timer.TT := 1, [33].Timer.EN := 1, [33].Timer.TT := 1, [34].Timer.EN := 1, [34].Timer.TT := 1, [35].Timer.EN := 1, [35].Timer.TT := 1, [36].Timer.EN := 1, [36].Timer.TT := 1, [37].Timer.EN := 1, [37].Timer.TT := 1, [38].Timer.EN := 1, [38].Timer.TT := 1, [39].Timer.EN := 1, [39].Timer.TT := 1, [40].Timer.EN := 1, [40].Timer.TT := 1, [41].Timer.EN := 1, [41].Timer.TT := 1, [42].Timer.EN := 1, [42].Timer.TT := 1, [43].Timer.EN := 1, [43].Timer.TT := 1, [44].Timer.EN := 1, [44].Timer.TT := 1, [45].Timer.EN := 1, [45].Timer.TT := 1, [46].Timer.EN := 1, [46].Timer.TT := 1, [47].Timer.EN := 1, [47].Timer.TT := 1, [48].Timer.EN := 1, [48].Timer.TT := 1, [49].Timer.EN := 1, [49].Timer.TT := 1,
        [50].Timer.EN := 1, [50].Timer.TT := 1, [51].Timer.EN := 1, [51].Timer.TT := 1, [52].Timer.EN := 1, [52].Timer.TT := 1, [53].Timer.EN := 1, [53].Timer.TT := 1, [54].Timer.EN := 1, [54].Timer.TT := 1, [55].Timer.EN := 1, [55].Timer.TT := 1, [56].Timer.EN := 1, [56].Timer.TT := 1, [57].Timer.EN := 1, [57].Timer.TT := 1, [58].Timer.EN := 1, [58].Timer.TT := 1, [59].Timer.EN := 1, [59].Timer.TT := 1, [60].Timer.EN := 1, [60].Timer.TT := 1, [61].Timer.EN := 1, [61].Timer.TT := 1, [62].Timer.EN := 1, [62].Timer.TT := 1, [63].Timer.EN := 1, [63].Timer.TT := 1, [64].Timer.EN := 1, [64].Timer.TT := 1, [65].Timer.EN := 1, [65].Timer.TT := 1, [66].Timer.EN := 1, [66].Timer.TT := 1, [67].Timer.EN := 1, [67].Timer.TT := 1, [68].Timer.EN := 1, [68].Timer.TT := 1, [69].Timer.EN := 1, [69].Timer.TT := 1, [70].Timer.EN := 1, [70].Timer.TT := 1, [71].Timer.EN := 1, [71].Timer.TT := 1, [72].Timer.EN := 1, [72].Timer.TT := 1, [73].Timer.EN := 1, [73].Timer.TT := 1, [74].Timer.EN := 1, [74].Timer.TT := 1, [75].Timer.EN := 1, [75].Timer.TT := 1, [76].Timer.EN := 1, [76].Timer.TT := 1, [77].Timer.EN := 1, [77].Timer.TT := 1, [78].Timer.EN := 1, [78].Timer.TT := 1, [79].Timer.EN := 1, [79].Timer.TT := 1,
        [80].Timer.EN := 1, [80].Timer.TT := 1, [81].Timer.EN := 1, [81].Timer.TT := 1, [82].Timer.EN := 1, [82].Timer.TT := 1, [83].Timer.EN := 1, [83].Timer.TT := 1, [84].Timer.EN := 1, [84].Timer.TT := 1, [85].Timer.EN := 1, [85].Timer.TT := 1, [86].Timer.EN := 1, [86].Timer.TT := 1, [87].Timer.EN := 1, [87].Timer.TT := 1, [88].Timer.EN := 1, [88].Timer.TT := 1, [89].Timer.EN := 1, [89].Timer.TT := 1, [90].Timer.EN := 1, [90].Timer.TT := 1, [91].Timer.EN := 1, [91].Timer.TT := 1, [92].Timer.EN := 1, [92].Timer.TT := 1, [93].Timer.EN := 1, [93].Timer.TT := 1, [94].Timer.EN := 1, [94].Timer.TT := 1, [95].Timer.EN := 1, [95].Timer.TT := 1, [96].Timer.EN := 1, [96].Timer.TT := 1, [97].Timer.EN := 1, [97].Timer.TT := 1, [98].Timer.EN := 1, [98].Timer.TT := 1, [99].Timer.EN := 1, [99].Timer.TT := 1);
   MQTT_OUT_B : DINT[100];
   MQTT_OUT_BOOL : UDT_MQTT_DINT[100] := ([0].Message := 2244, [0].RawData := 2244);
   MQTT_OUT_DINT : DINT[100] := ([0] := 36375, [1] := 236375, [2] := 5375);
   MSG_MTR07 : MESSAGE;
        MessageParameters(ServiceCode := 16#0032, LocalElement := motorReadReqs.Param_1_64[0], DestinationTag := M07_Params.Param_1_64[0], ...)
   MSG_MTR07_01 : MESSAGE;
        MessageParameters(ServiceCode := 16#0032, LocalElement := motorReadReqs.Param_65_128[0], DestinationTag := M07_Params.Param_65_128[0], ...)
   MSG_MTR07_02 : MESSAGE;
        MessageParameters(ServiceCode := 16#0032, LocalElement := motorReadReqs.Param_129_192[0], DestinationTag := M07_Params.Param_129_192[0], ...)
   MSG_MTR07_03 : MESSAGE;
        MessageParameters(ServiceCode := 16#0032, LocalElement := motorReadReqs.Param_193_256[0], DestinationTag := M07_Params.Param_193_256[0], ...)
   MSG_MTR07_04 : MESSAGE;
        MessageParameters(ServiceCode := 16#0032, LocalElement := motorReadReqs.Param_257_320[0], DestinationTag := M07_Params.Param_257_320[0], ...)
   MSG_MTR07_05 : MESSAGE;
        MessageParameters(ServiceCode := 16#0032, LocalElement := motorReadReqs.Param_321_384[0], DestinationTag := M07_Params.Param_321_384[0], ...)
   MSG_MTR07_06 : MESSAGE;
        MessageParameters(ServiceCode := 16#0032, LocalElement := motorReadReqs.Param_385_448[0], DestinationTag := M07_Params.Param_385_448[0], ...)
   MSG_MTR07_07 : MESSAGE;
        MessageParameters(ServiceCode := 16#0032, LocalElement := motorReadReqs.Param_449_512[0], DestinationTag := M07_Params.Param_449_512[0], ...)
   MSG_MTR07_08 : MESSAGE;
        MessageParameters(ServiceCode := 16#0032, LocalElement := motorReadReqs.Param_513_576[0], DestinationTag := M07_Params.Param_513_576[0], ...)
   MSG_MTR07_09 : MESSAGE;
        MessageParameters(ServiceCode := 16#0032, LocalElement := motorReadReqs.Param_577_640[0], DestinationTag := M07_Params.Param_577_640[0], ...)
   MSG_MTR07_10 : MESSAGE;
        MessageParameters(ServiceCode := 16#0032, LocalElement := motorReadReqs.Param_641_704[0], DestinationTag := M07_Params.Param_641_704[0], ...)
   MSG_MTR07_11 : MESSAGE;
        MessageParameters(ServiceCode := 16#0032, LocalElement := motorReadReqs.Param_705_768[0], DestinationTag := M07_Params.Param_705_768[0], ...)
   MTR1 : udtVariableSpeedMotor := (Ready := 1, FwdAct := 1, Avl[2] := 1);
   MTR_Speed : REAL[100];
   Pal_D : DINT[100] := ([0] := 2244, [1] := 9, [2] := 16);
        [0].1   // Palletizer Infeed - Stop PB
        [0].10   // Palletizer Discharge - Stop PB
        [0].12   // Palletizer Discharge - Full Pallet Ready
        [0].2   // Palletizer Infeed - Enabled Status
        [0].4   // Palletizer Robot - Start PB
        [0].7   // Palletizer Robot - Pick Up Cases
        [0].5   // Palletizer Robot - Stop PB
        [0].0   // Palletizer Infeed - Start PB
        [0].3   // Palletizer Infeed - Full Status
        [0].8   // Palletizer Robot - Cases On Arm
        [0].9   // Palletizer Discharge - Start PB
        [0].6   // Palletizer Robot - Enabled Status
        [0].11   // Palletizer Discharge - Running Status
   Pal_T : TIMER[100] := ([0].PRE := 1000, [0].ACC := 320, [0].EN := 1, [0].TT := 1, [1].PRE := 4268, [1].ACC := 1320, [1].EN := 1, [1].TT := 1, [2].PRE := 6639, [3].PRE := 7587);
   readReq1 : INT[2];
   readRes1 : INT[2] := ([0] := -32768, [1] := 22);
   scanTime_G : DINT := 233;
   ScanTimeMax : DINT := 609;
   ScanTimeMin : DINT := 220;
   SimulatedAssets_v01 : Asset_Data_v01_01[20] := ([0].machineState := 78, [0].currentProductionSpeed := 78);
   SolisPLC_B_IN_0 : BOOL;   // Start PB
   SolisPLC_B_IN_1 : BOOL := 1;   // Stop PB
   SolisPLC_B_IN_10 : BOOL;   // System 2 - Palletizer Infeed Stop Sensor
   SolisPLC_B_IN_11 : BOOL;   // MC - Start PB
   SolisPLC_B_IN_12 : BOOL := 1;   // MC - Stop PB
   SolisPLC_B_IN_13 : BOOL := 1;   // MC - Toggle Position 0
   SolisPLC_B_IN_14 : BOOL;   // MC - Toggle Position 1
   SolisPLC_B_IN_15 : BOOL;   // MCO - Belt 2 Part Detected
   SolisPLC_B_IN_16 : BOOL;   // MCO - Belt 1 Part Detected
   SolisPLC_B_IN_2 : BOOL;   // Box Present Photo Eye [BLOCKED]
   SolisPLC_B_IN_3 : BOOL;   // Box Wide Photo Eye [BLOCKED]
   SolisPLC_B_IN_4 : BOOL;   // Pivot Arm Sensor
   SolisPLC_B_IN_5 : BOOL;
   SolisPLC_B_IN_6 : BOOL;   // System 2 - Start Push Button
   SolisPLC_B_IN_7 : BOOL := 1;   // System 2 - Stop Push Button
   SolisPLC_B_IN_8 : BOOL;   // System 2 - Palletizer Infeed Sensor
   SolisPLC_B_IN_9 : BOOL;   // System 2 - Case Packer BackUp Sensor
   SolisPLC_B_OUT_0 : BOOL;   // Green Indicator
   SolisPLC_B_OUT_1 : BOOL := 1;   // Red Indicator
   SolisPLC_B_OUT_10 : BOOL;   // MC - Discharge Conveyor RUN
   SolisPLC_B_OUT_11 : BOOL;   // MC - Robot Cell / CNC RUN
   SolisPLC_B_OUT_12 : BOOL;   // MC - Machining Center Produce Lids
   SolisPLC_B_OUT_13 : BOOL;
   SolisPLC_B_OUT_14 : BOOL;
   SolisPLC_B_OUT_15 : BOOL;
   SolisPLC_B_OUT_16 : BOOL;   // MCO - Belt 1 Clamp
   SolisPLC_B_OUT_17 : BOOL;   // MCO - Belt 2 Clamp
   SolisPLC_B_OUT_18 : BOOL;   // MCO - Pivot
   SolisPLC_B_OUT_19 : BOOL;   // MCO - Grabber
   SolisPLC_B_OUT_2 : BOOL;   // Belt Conveyor 1 Run
   SolisPLC_B_OUT_20 : BOOL;   // MCO - Place X Axis
   SolisPLC_B_OUT_21 : BOOL;   // MCO - Place Z Axis
   SolisPLC_B_OUT_22 : BOOL;   // MCO - Belt 2 Raise
   SolisPLC_B_OUT_23 : BOOL;
   SolisPLC_B_OUT_3 : BOOL;   // Belt Conveyor 2 Run
   SolisPLC_B_OUT_4 : BOOL;   // Pivot Arm [TURN]
   SolisPLC_B_OUT_5 : BOOL;
   SolisPLC_B_OUT_6 : BOOL := 1;   // System 2 - Case Packer Enabled
   SolisPLC_B_OUT_7 : BOOL;   // System 2 - Case Packer Discharge Conveyor 1
   SolisPLC_B_OUT_8 : BOOL;   // System 2 - Palletizer Infeed Roller UP
   SolisPLC_B_OUT_9 : BOOL;   // MC - Infeed Conveyor RUN
   SolisPLC_F_IN_0 : REAL;
   SolisPLC_F_OUT_0 : REAL;   // System 2 - Palletizer Infeed Prior to Stop Conveyor
   SolisPLC_F_OUT_1 : REAL;   // System 2 - Palletizer Infeed After Stop Conveyor
   SolisPLC_I_OUT_0 : INT := 513;
   SolisPLC_I_OUT_1 : INT := 183;   // Wide Box Counter
   SolisPLC_I_OUT_2 : INT := 201;   // Narrow Box Counter
   SolisPLC_INT_IN_0 : INT;
   SolisPLC_INT_IN_1 : INT;
   SolisPLC_INT_OUT_0 : INT;
   SolisPLC_INT_OUT_1 : INT;
   Sys_Timer : TIMER[100] := ([0].PRE := 100000, [0].ACC := 36567, [0].EN := 1, [0].TT := 1, [1].PRE := 500000, [1].ACC := 236567, [1].EN := 1, [1].TT := 1, [2].PRE := 11000, [2].ACC := 5567, [2].EN := 1, [2].TT := 1);
   VFD_07 : udtVariableSpeedMotor;
   VFD_07_01 : MESSAGE;
        MessageParameters(ServiceCode := 16#0032, LocalElement := M07_readReq[0], DestinationTag := M07_readRes[0], ...)
   VFD_07_01b : MESSAGE;
        MessageParameters(ServiceCode := 16#0032, LocalElement := readReq1[0], DestinationTag := readRes1[0], ...)
   VladsExperiment1 : MUTING_TWO_SENSOR_ASYM;
   VladsFirstArray_B : BOOL[32];
   VladsFirstBoolean : BOOL := 1;
   VladsFirstCounter : COUNTER;
   VladsFirstInteger : INT := 120;
   VladsFirstPID : PID;
   VladsFirstREAL : REAL := 120.64;
   VladsFirstTime : TIMER;
   VladsSecondArray_B : BOOL[128];   // My Production Valves on Line 3
        [1]   // Vlave2
        [0]   // Valve 1
        [2]   // Valve 3
   VladsThirdArray_T : TIMER[10];
END_VAR

PROGRAM Communication   (* main routine _01_Main *)
VAR
   BOOL : BOOL[64];
   BOOL2 : DINT;
   ind1 : DINT;
   ind2 : DINT := 63;
   index : DINT := 64;
   MTR07_Read : DINT;
   MTR07_ReadNow : BOOL;
   T_DINT : DINT[20];
   T_MSG : TIMER := (PRE := 1000, ACC := 633, EN := 1, TT := 1);
   value : DINT := 768;
END_VAR

ROUTINE _01_Main   (* ladder *)
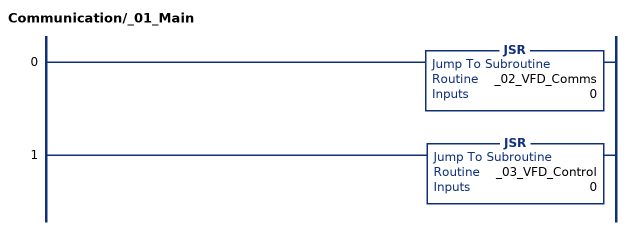
   0: JSR(_02_VFD_Comms,0);
   1: JSR(_03_VFD_Control,0);
END_ROUTINE

ROUTINE _02_VFD_Comms   (* ladder *)
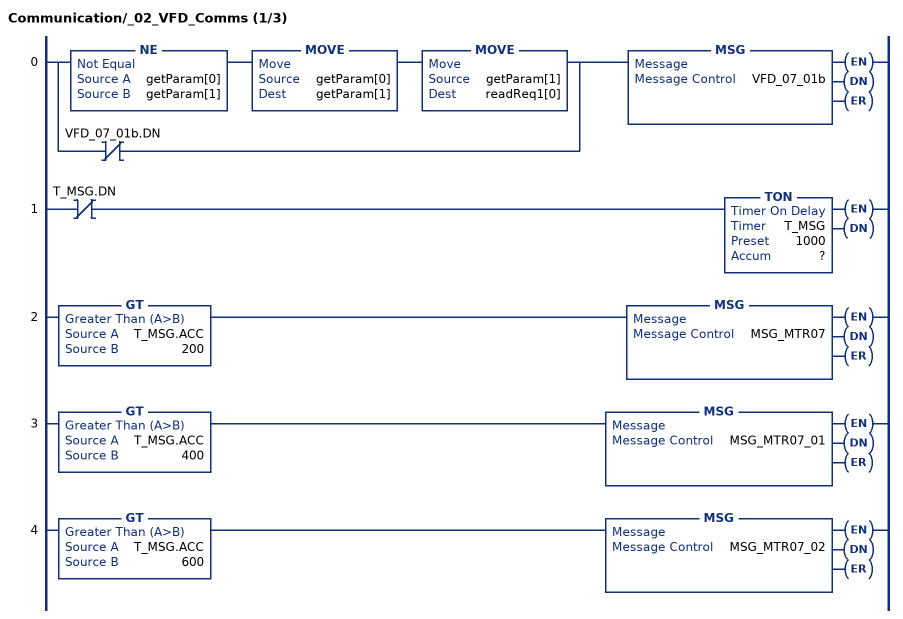
   0: [NE(getParam[0],getParam[1]) MOVE(getParam[0],getParam[1]) MOVE(getParam[1],readReq1[0]) ,XIO(VFD_07_01b.DN) ]MSG(VFD_07_01b);
   1: XIO(T_MSG.DN)TON(T_MSG,?,?);
   2: GT(T_MSG.ACC,200)MSG(MSG_MTR07);
   3: GT(T_MSG.ACC,400)MSG(MSG_MTR07_01);
   4: GT(T_MSG.ACC,600)MSG(MSG_MTR07_02);
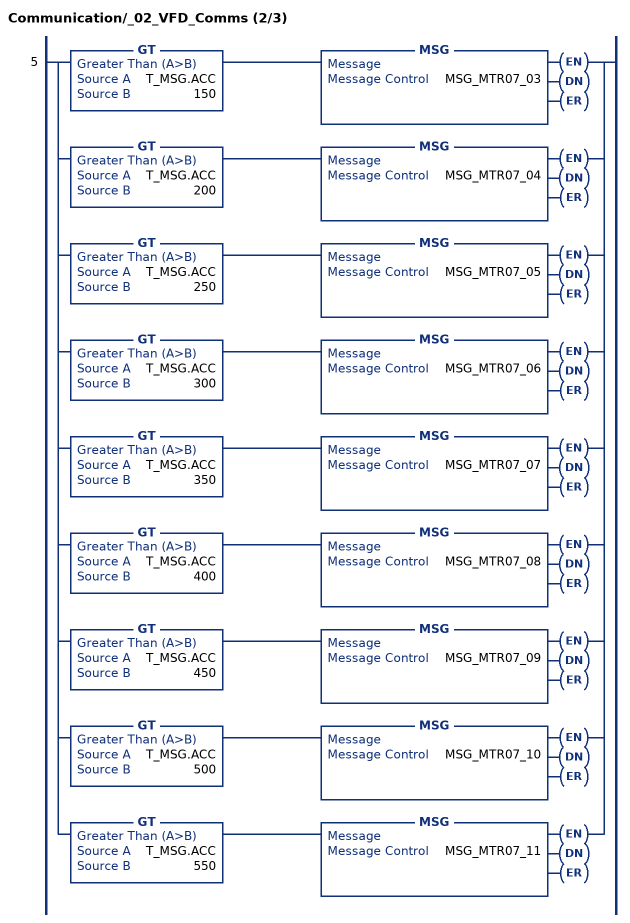
   5: [GT(T_MSG.ACC,150) MSG(MSG_MTR07_03) ,GT(T_MSG.ACC,200) MSG(MSG_MTR07_04) ,GT(T_MSG.ACC,250) MSG(MSG_MTR07_05) ,GT(T_MSG.ACC,300) MSG(MSG_MTR07_06) ,GT(T_MSG.ACC,350) MSG(MSG_MTR07_07) ,GT(T_MSG.ACC,400) MSG(MSG_MTR07_08) ,GT(T_MSG.ACC,450) MSG(MSG_MTR07_09) ,GT(T_MSG.ACC,500) MSG(MSG_MTR07_10) ,GT(T_MSG.ACC,550) MSG(MSG_MTR07_11) ];
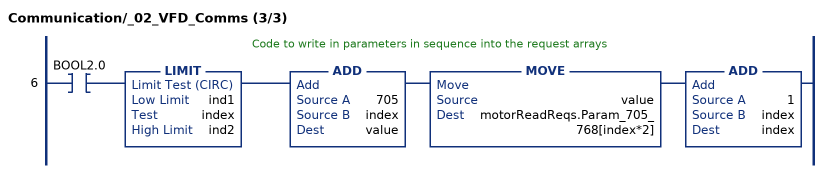
   // Code to write in parameters in sequence into the request arrays
   6: XIC(BOOL2.0)LIMIT(ind1,index,ind2)ADD(705,index,value)MOVE(value,motorReadReqs.Param_705_768[index*2])ADD(1,index,index);
END_ROUTINE
